FUNCTION_BLOCK HighTemperatureHeatingNetwork
VAR_INPUT
END_VAR
VAR_OUTPUT
END_VAR
VAR
END_VAR

END_FUNCTION_BLOCK

(* stored: Version 1.1.0.1, ProductVersion 3.1.4024.10
   POU HighTemperatureHeatingNetwork: Id {eb098d9a-ed09-496e-a742-15a3d3e6a2b2}, SpecialFunc None *)
